(* IEC 61131-3 sources: eCockpitGit/test_project/src/%F%00 Library/%F%Common Functions/%F%Bits/%F%Bit Set, 3 files *)

(* ---- %POU%FU_bBitSet.st ---- *)
//This function sets the bit value from a variable
// |**Version**|**Author**| **Date** |**Changes**                                                                                                            |
// | 1         | NSN      | 11-01-19 | Creation                                                                                                              |
FUNCTION FU_bBitSet : BOOL
VAR_IN_OUT
	bVar	:BYTE;		//The value to work with
END_VAR
VAR_INPUT
	bIndex	:BYTE;		//Which bit to get
	xVal	:BOOL;		//What to set the bit to
END_VAR
(*%!%__DELIMITER__%!%*)
bVar		:=		(bVar AND NOT(SHL(TO_BYTE(1),bIndex))) OR (SHL(TO_BYTE(xVal),bIndex));

(* ---- %POU%FU_dwBitSet.st ---- *)
//This function sets the bit value from a variable
// |**Version**|**Author**| **Date** |**Changes**
// | 1         | NSN      | 11-01-19 | Creation
FUNCTION FU_dwBitSet : BOOL
VAR_IN_OUT
	dbVar	:DWORD;		//The value to work with
END_VAR
VAR_INPUT
	bIndex		:BYTE;		//Which bit to get
	xVal		:BOOL;		//What to set the bit to
END_VAR
(*%!%__DELIMITER__%!%*)
dbVar		:=		(dbVar AND NOT(SHL(TO_DWORD(1),bIndex))) OR (SHL(TO_DWORD(xVal),bIndex));

(* ---- %POU%FU_wBitSet.st ---- *)
//This function sets the bit value from a variable
// |**Version**|**Author**| **Date** |**Changes**
// | 1         | NSN      | 11-01-19 | Creation
FUNCTION FU_wBitSet : BOOL
VAR_IN_OUT
	bVar	:WORD;		//The value to work with
END_VAR
VAR_INPUT
	bIndex	:BYTE;		//Which bit to get
	xVal	:BOOL;		//What to set the bit to
END_VAR
(*%!%__DELIMITER__%!%*)
bVar		:=		(bVar AND NOT(SHL(TO_WORD(1),bIndex))) OR (SHL(TO_WORD(xVal),bIndex));
